FUNCTION_BLOCK xrot_c
VAR_INPUT
    ix0: DINT;
    iy0: DINT;
    c: LREAL;
    b_s: LREAL;
END_VAR
VAR_IN_OUT
    x: ARRAY [0..29] OF LREAL;
END_VAR
VAR_TEMP
    k: DINT;
    temp_tmp: DINT;
    temp_tmp_0: LREAL;
    temp_tmp_1: DINT;
    temp_tmp_2: LREAL;
END_VAR

FOR k := 0 TO 5 DO 
    temp_tmp := (iy0 + k) - 1;
    temp_tmp_0 := x[temp_tmp];
    temp_tmp_1 := (ix0 + k) - 1;
    temp_tmp_2 := x[temp_tmp_1];
    x[temp_tmp] := (temp_tmp_0 * c) - (temp_tmp_2 * b_s);
    x[temp_tmp_1] := (temp_tmp_2 * c) + (temp_tmp_0 * b_s);
END_FOR;

END_FUNCTION_BLOCK

(* stored: Version 1.1.0.1, ProductVersion 3.1.4024.12
   POU xrot_c: Id {a3e3d615-b8a7-4d0c-bc0e-3f910ed79365}, SpecialFunc None *)
